PROGRAM MAIN
VAR

	IN_FUNZIONE: BOOL;
	IN_SMISTAMENTO: BOOL;
	TON_BIANCO: TON;
	TON_NERO: TON;
	PEZZO_BIANCO: BOOL;
	PEZZO_NERO: BOOL;
	IN_TIMBRATURA: BOOL;
	TON_TIMBRATURA_1: TON;
	TON_TIMBRATURA_2: TON;
	IN_FORATURA: BOOL;
	TON_FORATURA_1: TON;
	TON_FORATURA_2: TON;
END_VAR

GestionePulsantiSegnalazioni();
GestioneMotori();
GestioneSmistamento();
GestioneTimbratura();
GestioneForatura();
GestioneConteggio();

ACTION GestioneConteggio:
// NETWORK 1
END_ACTION

ACTION GestioneForatura:
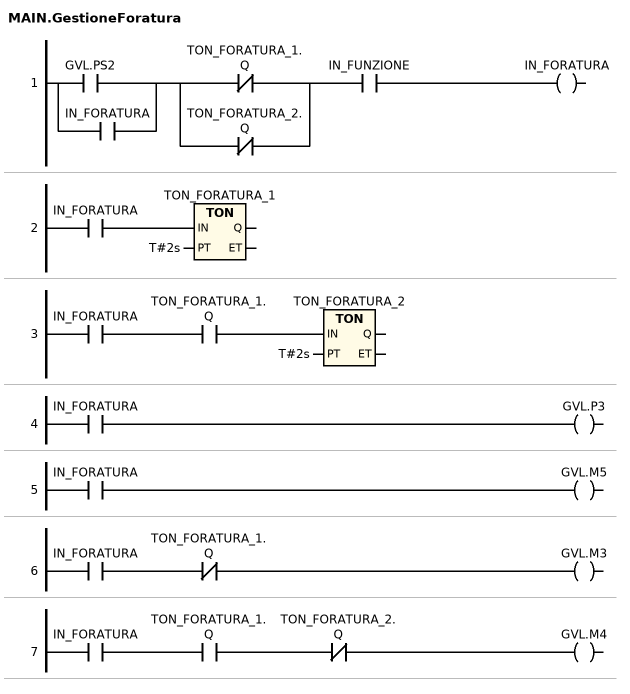
// NETWORK 1
IN_FORATURA := (GVL.PS2 OR IN_FORATURA) AND (NOT TON_FORATURA_1.Q OR NOT TON_FORATURA_2.Q) AND IN_FUNZIONE;

// NETWORK 2
TON_FORATURA_1(IN := IN_FORATURA, PT := T#2s); // TON

// NETWORK 3
TON_FORATURA_2(IN := IN_FORATURA AND TON_FORATURA_1.Q, PT := T#2s); // TON

// NETWORK 4
GVL.P3 := IN_FORATURA;

// NETWORK 5
GVL.M5 := IN_FORATURA;

// NETWORK 6
GVL.M3 := IN_FORATURA AND NOT TON_FORATURA_1.Q;

// NETWORK 7
GVL.M4 := IN_FORATURA AND TON_FORATURA_1.Q AND NOT TON_FORATURA_2.Q;
END_ACTION

ACTION GestioneMotori:
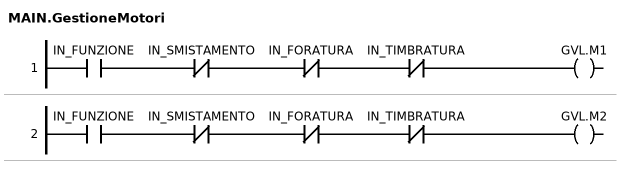
// NETWORK 1
GVL.M1 := IN_FUNZIONE AND NOT IN_SMISTAMENTO AND NOT IN_FORATURA AND NOT IN_TIMBRATURA;

// NETWORK 2
GVL.M2 := IN_FUNZIONE AND NOT IN_SMISTAMENTO AND NOT IN_FORATURA AND NOT IN_TIMBRATURA;
END_ACTION

ACTION GestionePulsantiSegnalazioni:
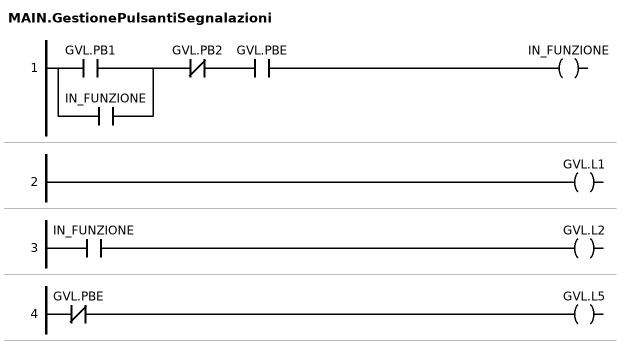
// NETWORK 1
IN_FUNZIONE := (GVL.PB1 OR IN_FUNZIONE) AND NOT GVL.PB2 AND GVL.PBE;

// NETWORK 2
GVL.L1 := TRUE;

// NETWORK 3
GVL.L2 := IN_FUNZIONE;

// NETWORK 4
GVL.L5 := NOT GVL.PBE;
END_ACTION

ACTION GestioneSmistamento:
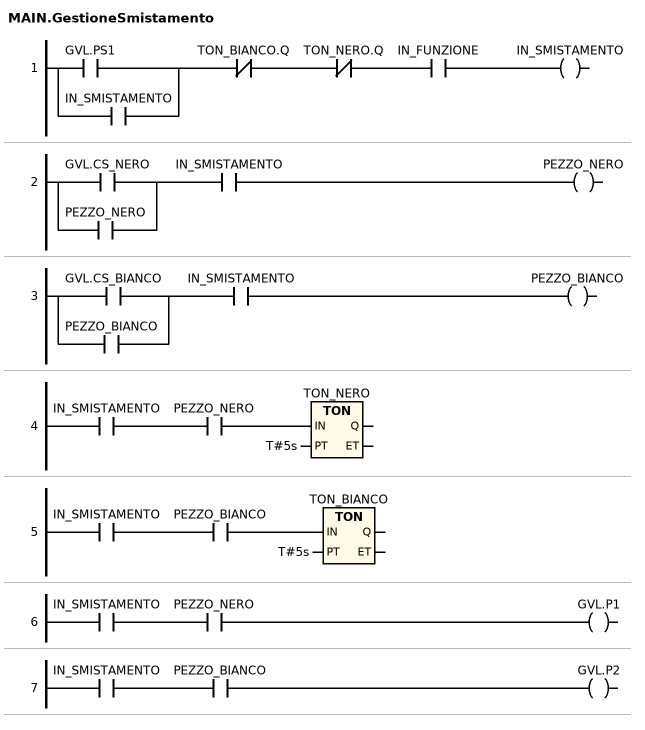
// NETWORK 1
IN_SMISTAMENTO := (GVL.PS1 OR IN_SMISTAMENTO) AND NOT TON_BIANCO.Q AND NOT TON_NERO.Q AND IN_FUNZIONE;

// NETWORK 2
PEZZO_NERO := (GVL.CS_NERO OR PEZZO_NERO) AND IN_SMISTAMENTO;

// NETWORK 3
PEZZO_BIANCO := (GVL.CS_BIANCO OR PEZZO_BIANCO) AND IN_SMISTAMENTO;

// NETWORK 4
TON_NERO(IN := IN_SMISTAMENTO AND PEZZO_NERO, PT := T#5s); // TON

// NETWORK 5
TON_BIANCO(IN := IN_SMISTAMENTO AND PEZZO_BIANCO, PT := T#5s); // TON

// NETWORK 6
GVL.P1 := IN_SMISTAMENTO AND PEZZO_NERO;

// NETWORK 7
GVL.P2 := IN_SMISTAMENTO AND PEZZO_BIANCO;
END_ACTION

ACTION GestioneTimbratura:
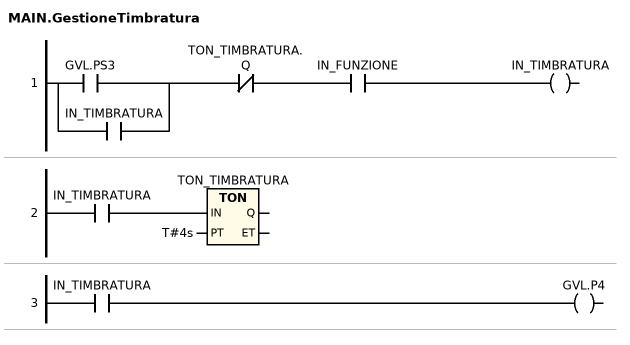
// NETWORK 1
IN_TIMBRATURA := (GVL.PS3 OR IN_TIMBRATURA) AND NOT TON_TIMBRATURA.Q AND IN_FUNZIONE;

// NETWORK 2
TON_TIMBRATURA(IN := IN_TIMBRATURA, PT := T#4s); // TON

// NETWORK 3
GVL.P4 := IN_TIMBRATURA;
END_ACTION

END_PROGRAM

(* stored: Version 1.1.0.1, ProductVersion 3.1.4024.12
   POU MAIN: Id {77ce3c58-9155-42f5-9eb6-c02febfddbf9}, SpecialFunc None
   Action GestioneConteggio: Id {619b20d3-e452-44f5-b626-dfa96b8409ac}
   Action GestioneForatura: Id {231e95f2-6121-4dbc-89e6-afb7e53183f4}
   Action GestioneMotori: Id {9e464890-6681-41a5-8f39-3082d5bac0ef}
   Action GestionePulsantiSegnalazioni: Id {3f00a759-f8d0-455e-af78-03f29b3994ec}
   Action GestioneSmistamento: Id {6f07de2f-68ba-41e8-a08f-d2eacd4f38eb}
   Action GestioneTimbratura: Id {12208fa5-515e-473c-96cd-01596b797502} *)
